{attribute 'GeneratedUsingTerminal: EJ1957-0000-0017'}
{attribute addProperty BoxType "EJ1957-0000-0017"}
{attribute addProperty Id "Module_1_FSOEModule_1_FSOE_9FCACE1432Module_2_FSOUTModule_2_FSOUT_5A5AEBA44Module_3_DEVICEIOModule_3_DEVICEIO_5FA6B4E72Module_4_FSLOGICModule_4_FSLOGIC_DEAB45222WcStateAT %I*WcState_B516A2644InfoDataAT %I*InfoData_94A18F5E2"}
{attribute addProperty CRC "3393175183"}
{attribute addProperty Size "46"}
TYPE EJ1957_CA3FBE8F EXTENDS EtcSlaveTerminalBase_947E5A46 :
STRUCT
	{attribute addProperty Name "Module_1_FSOE"}
	Module_1_FSOE : Module_1_FSOE_9FCACE14;
	{attribute addProperty Name "Module_2_FSOUT"}
	Module_2_FSOUT : Module_2_FSOUT_5A5AEBA4;
	{attribute addProperty Name "Module_3_DEVICEIO"}
	Module_3_DEVICEIO : Module_3_DEVICEIO_5FA6B4E7;
	{attribute addProperty Name "Module_4_FSLOGIC"}
	Module_4_FSLOGIC : Module_4_FSLOGIC_DEAB4522;
	{attribute addProperty Name "WcState"}
	WcState : WcState_B516A264;
	{attribute addProperty Name "InfoData"}
	InfoData : InfoData_94A18F5E;
END_STRUCT
END_TYPE

(* stored: Version 1.2.0.0, ProductVersion 3.1.4024.9
   DUT EJ1957_CA3FBE8F: Id {3edc3441-3923-4351-a4a4-4a564c8a4caa} *)
